{attribute 'GeneratedUsingTerminal: EM2042-0000-0016'}
{attribute addProperty BoxType "EM2042-0000-0016"}
{attribute addProperty Id "WcStateAT %I*BOOL1"}
{attribute addProperty CRC "187373305"}
{attribute addProperty Size "1"}
TYPE WcState_0B2B16F9 :
STRUCT
	{attribute addProperty Name "WcState"}
	WcState AT %I* : BOOL;
END_STRUCT
END_TYPE

(* stored: Version 1.2.0.0, ProductVersion 3.1.4024.11
   DUT WcState_0B2B16F9: Id {ff76cf35-0664-4c7f-bf73-3eb1879baf9b} *)
